{attribute 'GeneratedUsingTerminal: EP9128-0021-0016'}
{attribute addProperty BoxType "EP9128-0021-0016"}
{attribute addProperty Id "A_0007_EP9128_0021_0017A_0007_EP9128_0021_0017_AEE99380531A_0004_EP9128_0021_0016_2_EP9128_1021EP9128_1FC0878B2"}
{attribute addProperty CRC "2922841757"}
{attribute addProperty Size "533"}
TYPE A_0004_EP9128_0021_0016_AE37069D EXTENDS EP9128_1FC0878B :
STRUCT
	{attribute addProperty Name "A_0007_EP9128_0021_0017"}
	{attribute addProperty PreviousPort "A_0004(EP9128-0021-0016) : D"}
	A_0007_EP9128_0021_0017 : A_0007_EP9128_0021_0017_AEE99380;
	{attribute addProperty Name "A_0004_EP9128_0021_0016_2_EP9128_1021"}
	{attribute addProperty PreviousPort "A_0004(EP9128-0021-0016) : C"}
	A_0004_EP9128_0021_0016_2_EP9128_1021 : EP9128_1FC0878B;
END_STRUCT
END_TYPE

(* stored: Version 1.2.0.0, ProductVersion 3.1.4024.9
   DUT A_0004_EP9128_0021_0016_AE37069D: Id {b4188edf-27f0-4f0a-bd95-a89f19c308db} *)
